FUNCTION_BLOCK INTERNAL FB_WriteRepeatedFieldMessageTests EXTENDS FB_TestSuite
VAR
	fbWriteCtx		: FB_WriteContext;
	fbFoo   		: FB_Foo;
	stFoo           : ST_Foo;
	aBuffer 		: ARRAY[0..255] OF BYTE;
END_VAR

TEST(__POUNAME());


// Arrange
fbWriteCtx.FromBuffer(aBuffer);
stFoo.baz[0].value:= 42;
stFoo.baz[0].name:= 'foo';
stFoo.baz[1].value:= 6969;
stFoo.baz[1].name:= 'bar';
stFoo.baz[2].value:= 1337;
stFoo.baz[2].name:= 'baz';
F_SetMessageValue(F_ToAnyType(stFoo), fbFoo);

// Act 
fbFoo.WriteTo(fbWriteCtx);



// Assert



TEST_FINISHED_NAMED(__POUNAME());

END_FUNCTION_BLOCK

(* stored: Version 1.1.0.1
   POU FB_WriteRepeatedFieldMessageTests: Id {89bc8e78-f313-44c0-ab2f-dd749b8a02dd}, SpecialFunc None *)
